{attribute 'linkalways'} 
{attribute 'no_explicit_call' := 'This FB is a CLASS and must be accessed using methods or properties'}
{attribute 'enable_dynamic_creation'}
FUNCTION_BLOCK Node_F_VN_GetAt_ITcVnContainer EXTENDS VisionNode
VAR
    ipSrcContainer : _ITcVnContainer;
    ipDestContainer : _ITcVnContainer;
    nIndex : _ULINT(0);
    hrPrev : _HRESULT(S_OK);
    hresult : _HRESULT(S_OK);
END_VAR

METHOD PUBLIC  Clone : I_Node
VAR
	pNode : POINTER TO Node_F_VN_GetAt_ITcVnContainer;
END_VAR
pNode := __NEW(Node_F_VN_GetAt_ITcVnContainer);
Clone := pNode^;
END_METHOD

METHOD FB_init : BOOL
VAR_INPUT
	bInitRetains : BOOL; // if TRUE, the retain variables are initialized (warm start / cold start)
	bInCopyCode : BOOL;  // if TRUE, the instance afterwards gets moved into the copy code (online change)
END_VAR
AddInput('ipSrcContainer', ipSrcContainer);
AddInput('nIndex', nIndex);
AddInput('hrPrev', hrPrev);
AddOutput('ipDestContainer', ipDestContainer);
AddOutput('hresult',hresult);
END_METHOD

METHOD PROTECTED OnExecute : HRESULT
hresult.Value := F_VN_GetAt_ITcVnContainer(
    ipSrcContainer := ipSrcContainer.Value,
    ipDestContainer := ipDestContainer.Value,
    nIndex := nIndex.Value,
    hrPrev:= hrPrev.Value);
END_METHOD

METHOD PUBLIC PreExecutionCheck
VAR_INPUT
	Check : I_PreExecutionChecks;
END_VAR
IF FAILED(hrPrev.Value) THEN
    RETURN;
END_IF

Check.IsTrue(ipSrcContainer.IsValid, 'ipSrcContainer must be a valid container');
//TODO Check.IsTrue(ipSrcContainer.HasType( ??? ), 'ipSrcContainer contains incorrect type');
END_METHOD

END_FUNCTION_BLOCK

(* stored: Version 1.1.0.1, ProductVersion 3.1.4024.13
   POU Node_F_VN_GetAt_ITcVnContainer: Id {8ed8d91a-c872-4871-835f-90dc40093bd4}, SpecialFunc None
   Folder Constructor: Id {6856f3c3-94d0-40be-830a-ee629ded857a}
   Method Clone: Id {9e97bbdf-801c-42b5-a90f-7be710820a6b}
   Method FB_init: Id {656f031e-ed3a-4822-b020-02ec1c31e0d1}
   Method OnExecute: Id {7a0a19c3-a038-4576-b85a-e94c9e72f3bd}
   Method PreExecutionCheck: Id {48084579-9c4b-4ac9-b069-8984c9e01492} *)
